# EPICS substitutions: apps/mpodLvApp/Db/ftaglv.substitutions
file "db/mpod8008l.db" {
    pattern {HOST,CH,SCAN,PORT,DETALIAS}
  {"129.57.86.109",  "0","5 second","B_HW_LVFTAG_Sl0_Ch0","B_DET_FTC_LV_Q1Q4P"}
  {"129.57.86.109",  "1","5 second","B_HW_LVFTAG_Sl0_Ch1","B_DET_FTC_LV_Q1Q4N"}
  {"129.57.86.109",  "2","5 second","B_HW_LVFTAG_Sl0_Ch2","B_DET_FTC_LV_Q2Q3P"}
  {"129.57.86.109",  "3","5 second","B_HW_LVFTAG_Sl0_Ch3","B_DET_FTC_LV_Q2Q3N"}
}

#{"129.57.86.109",  "2","5 second","B_HW_LVFTAG_Sl0_Ch2","B_DET_FT_LV_Sl0_Ch2"}
#{"129.57.86.109",  "3","5 second","B_HW_LVFTAG_Sl0_Ch3","B_DET_FT_LV_Sl0_Ch3"}
#{"129.57.86.109",  "4","5 second","B_HW_LVFTAG_Sl0_Ch4","B_DET_FT_LV_Sl0_Ch4"}
#{"129.57.86.109",  "5","5 second","B_HW_LVFTAG_Sl0_Ch5","B_DET_FT_LV_Sl0_Ch5"}
#{"129.57.86.109",  "6","5 second","B_HW_LVFTAG_Sl0_Ch6","B_DET_FT_LV_Sl0_Ch6"}
#{"129.57.86.109",  "7","5 second","B_HW_LVFTAG_Sl0_Ch7","B_DET_FT_LV_Sl0_Ch7"}
#{"129.57.86.109","100","5 second","B_HW_LVFTAG_Sl1_Ch0","B_DET_FT_LV_Sl1_Ch0"}
#{"129.57.86.109","101","5 second","B_HW_LVFTAG_Sl1_Ch1","B_DET_FT_LV_Sl1_Ch1"}
#{"129.57.86.109","102","5 second","B_HW_LVFTAG_Sl1_Ch2","B_DET_FT_LV_Sl1_Ch2"}
#{"129.57.86.109","103","5 second","B_HW_LVFTAG_Sl1_Ch3","B_DET_FT_LV_Sl1_Ch3"}
#{"129.57.86.109","104","5 second","B_HW_LVFTAG_Sl1_Ch4","B_DET_FT_LV_Sl1_Ch4"}
#{"129.57.86.109","105","5 second","B_HW_LVFTAG_Sl1_Ch5","B_DET_FT_LV_Sl1_Ch5"}
#{"129.57.86.109","106","5 second","B_HW_LVFTAG_Sl1_Ch6","B_DET_FT_LV_Sl1_Ch6"}
#{"129.57.86.109","107","5 second","B_HW_LVFTAG_Sl1_Ch7","B_DET_FT_LV_Sl1_Ch7"}
#{"129.57.86.109","200","5 second","B_HW_LVFTAG_Sl2_Ch0","B_DET_FT_LV_Sl2_Ch0"}
#{"129.57.86.109","201","5 second","B_HW_LVFTAG_Sl2_Ch1","B_DET_FT_LV_Sl2_Ch1"}
#{"129.57.86.109","202","5 second","B_HW_LVFTAG_Sl2_Ch2","B_DET_FT_LV_Sl2_Ch2"}
#{"129.57.86.109","203","5 second","B_HW_LVFTAG_Sl2_Ch3","B_DET_FT_LV_Sl2_Ch3"}
#{"129.57.86.109","204","5 second","B_HW_LVFTAG_Sl2_Ch4","B_DET_FT_LV_Sl2_Ch4"}
#{"129.57.86.109","205","5 second","B_HW_LVFTAG_Sl2_Ch5","B_DET_FT_LV_Sl2_Ch5"}
#{"129.57.86.109","206","5 second","B_HW_LVFTAG_Sl2_Ch6","B_DET_FT_LV_Sl2_Ch6"}
#{"129.57.86.109","207","5 second","B_HW_LVFTAG_Sl2_Ch7","B_DET_FT_LV_Sl2_Ch7"}
